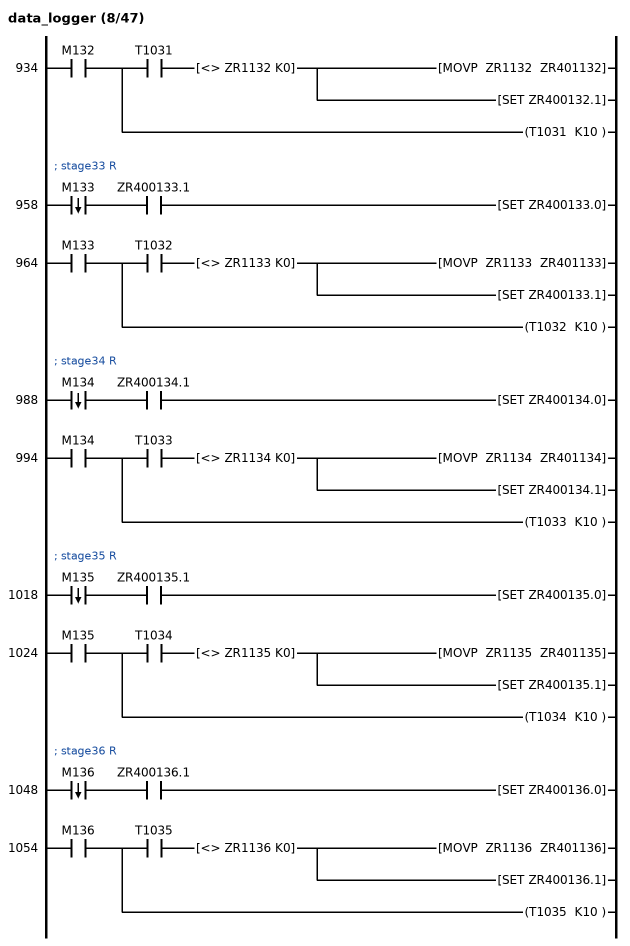
[picture p120: ladder of data_logger, rungs at steps 934 to 1054]
934   LD      M132
      MPS
      AND     T1031
      AND<>   ZR1132 K0
      MOVP    ZR1132 ZR401132
      SET     ZR400132.1
      MPP
      OUT     T1031 K10
; stage33 R
958   LDF     M133
      AND     ZR400133.1
      SET     ZR400133.0
964   LD      M133
      MPS
      AND     T1032
      AND<>   ZR1133 K0
      MOVP    ZR1133 ZR401133
      SET     ZR400133.1
      MPP
      OUT     T1032 K10
; stage34 R
988   LDF     M134
      AND     ZR400134.1
      SET     ZR400134.0
994   LD      M134
      MPS
      AND     T1033
      AND<>   ZR1134 K0
      MOVP    ZR1134 ZR401134
      SET     ZR400134.1
      MPP
      OUT     T1033 K10
; stage35 R
1018  LDF     M135
      AND     ZR400135.1
      SET     ZR400135.0
1024  LD      M135
      MPS
      AND     T1034
      AND<>   ZR1135 K0
      MOVP    ZR1135 ZR401135
      SET     ZR400135.1
      MPP
      OUT     T1034 K10
; stage36 R
1048  LDF     M136
      AND     ZR400136.1
      SET     ZR400136.0
1054  LD      M136
      MPS
      AND     T1035
      AND<>   ZR1136 K0
      MOVP    ZR1136 ZR401136
      SET     ZR400136.1
      MPP
      OUT     T1035 K10
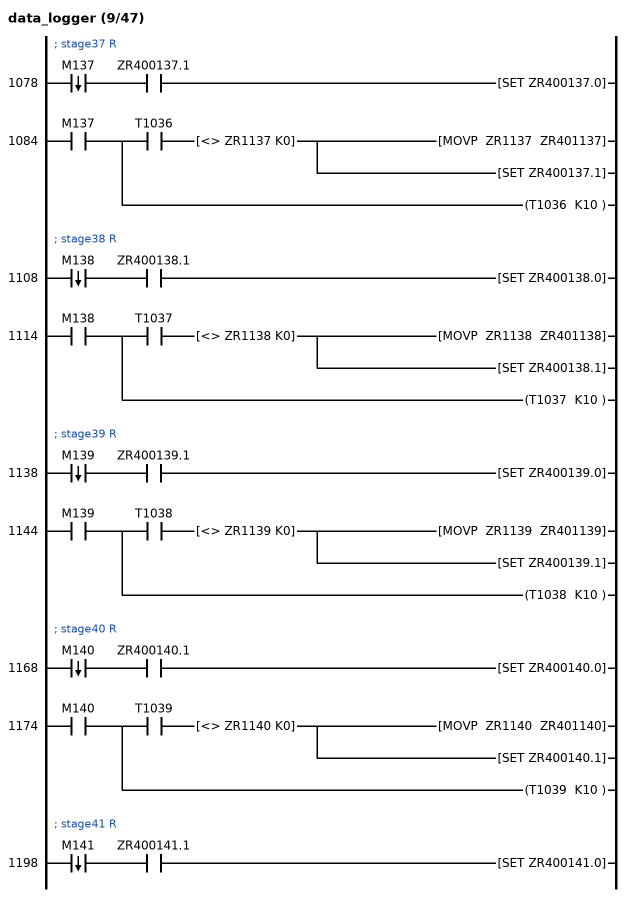
; stage37 R
1078  LDF     M137
      AND     ZR400137.1
      SET     ZR400137.0
1084  LD      M137
      MPS
      AND     T1036
      AND<>   ZR1137 K0
      MOVP    ZR1137 ZR401137
      SET     ZR400137.1
      MPP
      OUT     T1036 K10
; stage38 R
1108  LDF     M138
      AND     ZR400138.1
      SET     ZR400138.0
1114  LD      M138
      MPS
      AND     T1037
      AND<>   ZR1138 K0
      MOVP    ZR1138 ZR401138
      SET     ZR400138.1
      MPP
      OUT     T1037 K10
; stage39 R
1138  LDF     M139
      AND     ZR400139.1
      SET     ZR400139.0
1144  LD      M139
      MPS
      AND     T1038
      AND<>   ZR1139 K0
      MOVP    ZR1139 ZR401139
      SET     ZR400139.1
      MPP
      OUT     T1038 K10
; stage40 R
1168  LDF     M140
      AND     ZR400140.1
      SET     ZR400140.0
1174  LD      M140
      MPS
      AND     T1039
      AND<>   ZR1140 K0
      MOVP    ZR1140 ZR401140
      SET     ZR400140.1
      MPP
      OUT     T1039 K10
; stage41 R
1198  LDF     M141
      AND     ZR400141.1
      SET     ZR400141.0
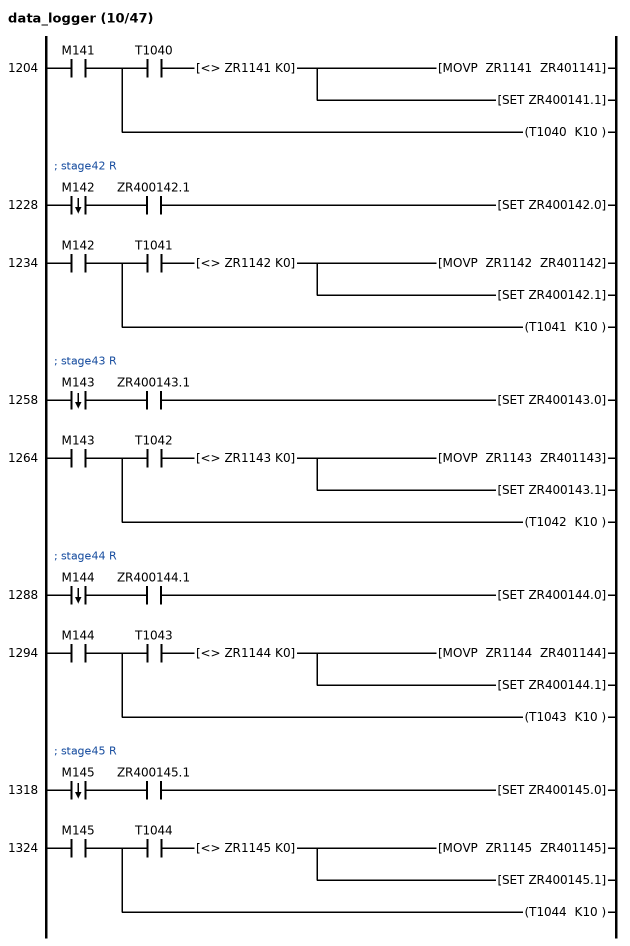
1204  LD      M141
      MPS
      AND     T1040
      AND<>   ZR1141 K0
      MOVP    ZR1141 ZR401141
      SET     ZR400141.1
      MPP
      OUT     T1040 K10
; stage42 R
1228  LDF     M142
      AND     ZR400142.1
      SET     ZR400142.0
1234  LD      M142
      MPS
      AND     T1041
      AND<>   ZR1142 K0
      MOVP    ZR1142 ZR401142
      SET     ZR400142.1
      MPP
      OUT     T1041 K10
; stage43 R
1258  LDF     M143
      AND     ZR400143.1
      SET     ZR400143.0
1264  LD      M143
      MPS
      AND     T1042
      AND<>   ZR1143 K0
      MOVP    ZR1143 ZR401143
      SET     ZR400143.1
      MPP
      OUT     T1042 K10
; stage44 R
1288  LDF     M144
      AND     ZR400144.1
      SET     ZR400144.0
1294  LD      M144
      MPS
      AND     T1043
      AND<>   ZR1144 K0
      MOVP    ZR1144 ZR401144
      SET     ZR400144.1
      MPP
      OUT     T1043 K10
; stage45 R
1318  LDF     M145
      AND     ZR400145.1
      SET     ZR400145.0
1324  LD      M145
      MPS
      AND     T1044
      AND<>   ZR1145 K0
      MOVP    ZR1145 ZR401145
      SET     ZR400145.1
      MPP
      OUT     T1044 K10
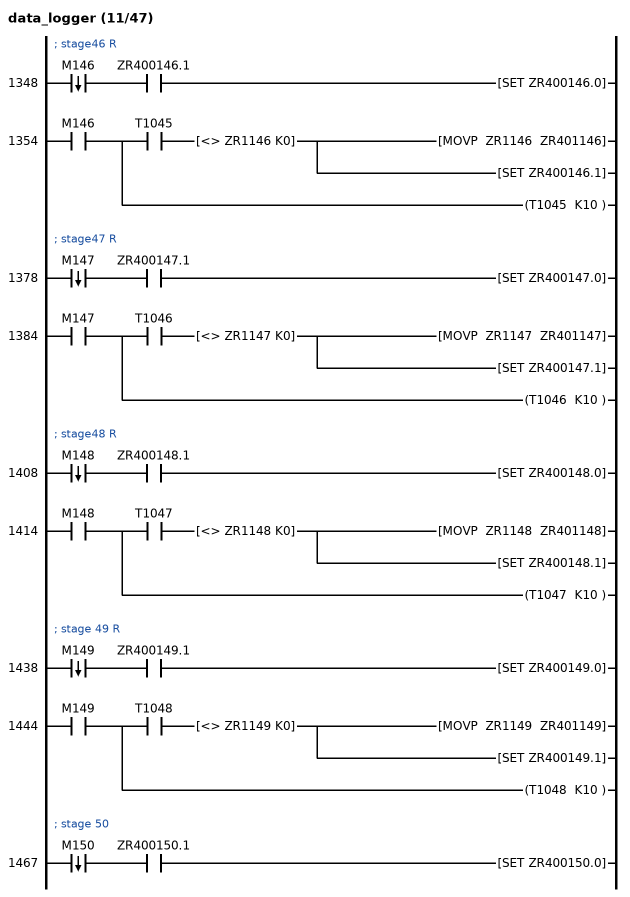
; stage46 R
1348  LDF     M146
      AND     ZR400146.1
      SET     ZR400146.0
1354  LD      M146
      MPS
      AND     T1045
      AND<>   ZR1146 K0
      MOVP    ZR1146 ZR401146
      SET     ZR400146.1
      MPP
      OUT     T1045 K10
; stage47 R
1378  LDF     M147
      AND     ZR400147.1
      SET     ZR400147.0
1384  LD      M147
      MPS
      AND     T1046
      AND<>   ZR1147 K0
      MOVP    ZR1147 ZR401147
      SET     ZR400147.1
      MPP
      OUT     T1046 K10
; stage48 R
1408  LDF     M148
      AND     ZR400148.1
      SET     ZR400148.0
1414  LD      M148
      MPS
      AND     T1047
      AND<>   ZR1148 K0
      MOVP    ZR1148 ZR401148
      SET     ZR400148.1
      MPP
      OUT     T1047 K10
; stage 49 R
1438  LDF     M149
      AND     ZR400149.1
      SET     ZR400149.0
1444  LD      M149
      MPS
      AND     T1048
      AND<>   ZR1149 K0
      MOVP    ZR1149 ZR401149
      SET     ZR400149.1
      MPP
      OUT     T1048 K10
; stage 50
1467  LDF     M150
      AND     ZR400150.1
      SET     ZR400150.0
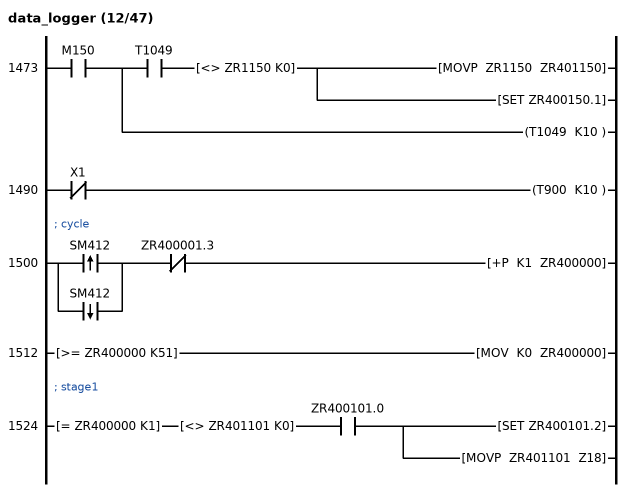
1473  LD      M150
      MPS
      AND     T1049
      AND<>   ZR1150 K0
      MOVP    ZR1150 ZR401150
      SET     ZR400150.1
      MPP
      OUT     T1049 K10
1490  LDI     X1
      OUT     T900 K10
; cycle
1500  LDP     SM412
      ORF     SM412
      ANI     ZR400001.3
      +P      K1 ZR400000
1512  LD>=    ZR400000 K51
      MOV     K0 ZR400000
; stage1
1524  LD=     ZR400000 K1
      AND<>   ZR401101 K0
      AND     ZR400101.0
      SET     ZR400101.2
      MOVP    ZR401101 Z18
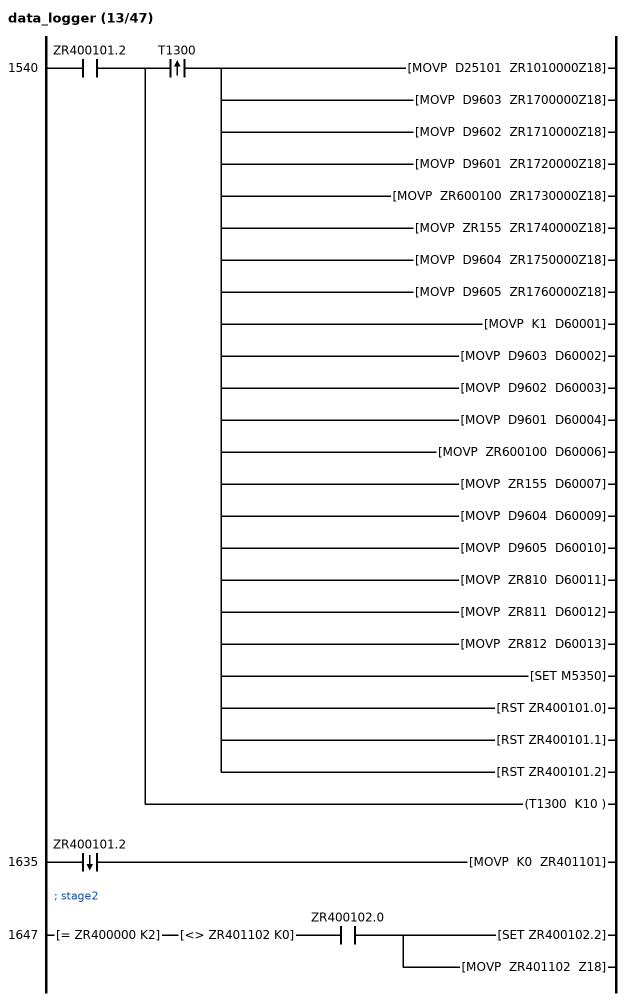
1540  LD      ZR400101.2
      MPS
      ANDP    T1300
      MOVP    D25101 ZR1010000Z18
      MOVP    D9603 ZR1700000Z18
      MOVP    D9602 ZR1710000Z18
      MOVP    D9601 ZR1720000Z18
      MOVP    ZR600100 ZR1730000Z18
      MOVP    ZR155 ZR1740000Z18
      MOVP    D9604 ZR1750000Z18
      MOVP    D9605 ZR1760000Z18
      MOVP    K1 D60001
      MOVP    D9603 D60002
      MOVP    D9602 D60003
      MOVP    D9601 D60004
      MOVP    ZR600100 D60006
      MOVP    ZR155 D60007
      MOVP    D9604 D60009
      MOVP    D9605 D60010
      MOVP    ZR810 D60011
      MOVP    ZR811 D60012
      MOVP    ZR812 D60013
      SET     M5350
      RST     ZR400101.0
      RST     ZR400101.1
      RST     ZR400101.2
      MPP
      OUT     T1300 K10
1635  LDF     ZR400101.2
      MOVP    K0 ZR401101
; stage2
1647  LD=     ZR400000 K2
      AND<>   ZR401102 K0
      AND     ZR400102.0
      SET     ZR400102.2
      MOVP    ZR401102 Z18
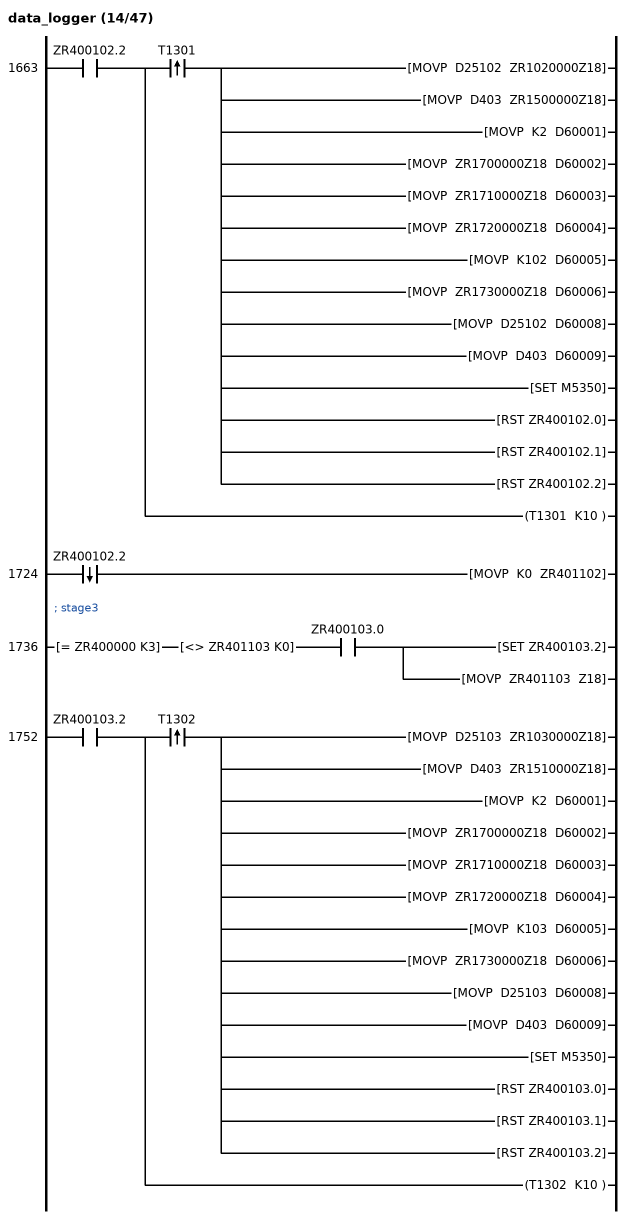
1663  LD      ZR400102.2
      MPS
      ANDP    T1301
      MOVP    D25102 ZR1020000Z18
      MOVP    D403 ZR1500000Z18
      MOVP    K2 D60001
      MOVP    ZR1700000Z18 D60002
      MOVP    ZR1710000Z18 D60003
      MOVP    ZR1720000Z18 D60004
      MOVP    K102 D60005
      MOVP    ZR1730000Z18 D60006
      MOVP    D25102 D60008
      MOVP    D403 D60009
      SET     M5350
      RST     ZR400102.0
      RST     ZR400102.1
      RST     ZR400102.2
      MPP
      OUT     T1301 K10
1724  LDF     ZR400102.2
      MOVP    K0 ZR401102
; stage3
1736  LD=     ZR400000 K3
      AND<>   ZR401103 K0
      AND     ZR400103.0
      SET     ZR400103.2
      MOVP    ZR401103 Z18
1752  LD      ZR400103.2
      MPS
      ANDP    T1302
      MOVP    D25103 ZR1030000Z18
      MOVP    D403 ZR1510000Z18
      MOVP    K2 D60001
      MOVP    ZR1700000Z18 D60002
      MOVP    ZR1710000Z18 D60003
      MOVP    ZR1720000Z18 D60004
      MOVP    K103 D60005
      MOVP    ZR1730000Z18 D60006
      MOVP    D25103 D60008
      MOVP    D403 D60009
      SET     M5350
      RST     ZR400103.0
      RST     ZR400103.1
      RST     ZR400103.2
      MPP
      OUT     T1302 K10
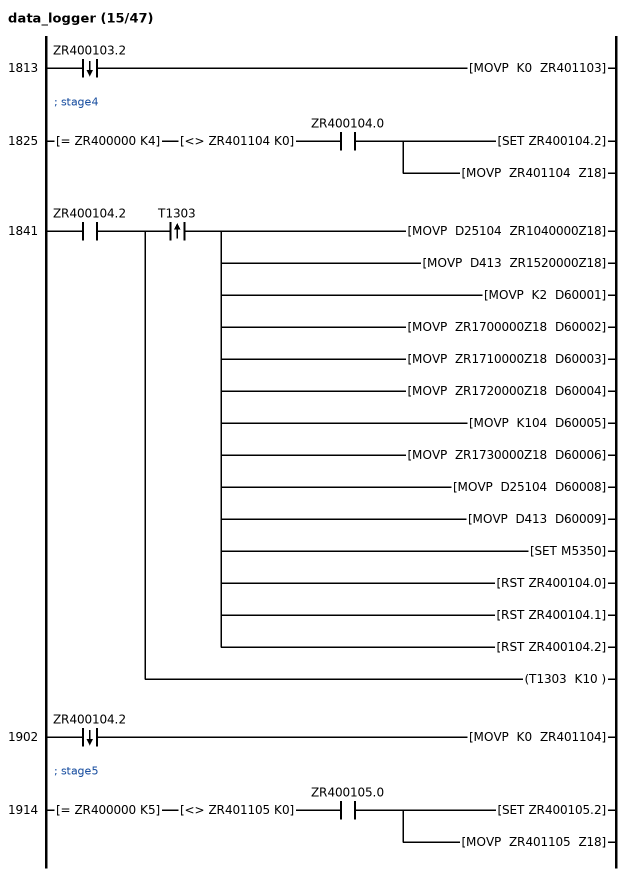
1813  LDF     ZR400103.2
      MOVP    K0 ZR401103
; stage4
1825  LD=     ZR400000 K4
      AND<>   ZR401104 K0
      AND     ZR400104.0
      SET     ZR400104.2
      MOVP    ZR401104 Z18
1841  LD      ZR400104.2
      MPS
      ANDP    T1303
      MOVP    D25104 ZR1040000Z18
      MOVP    D413 ZR1520000Z18
      MOVP    K2 D60001
      MOVP    ZR1700000Z18 D60002
      MOVP    ZR1710000Z18 D60003
      MOVP    ZR1720000Z18 D60004
      MOVP    K104 D60005
      MOVP    ZR1730000Z18 D60006
      MOVP    D25104 D60008
      MOVP    D413 D60009
      SET     M5350
      RST     ZR400104.0
      RST     ZR400104.1
      RST     ZR400104.2
      MPP
      OUT     T1303 K10
1902  LDF     ZR400104.2
      MOVP    K0 ZR401104
; stage5
1914  LD=     ZR400000 K5
      AND<>   ZR401105 K0
      AND     ZR400105.0
      SET     ZR400105.2
      MOVP    ZR401105 Z18
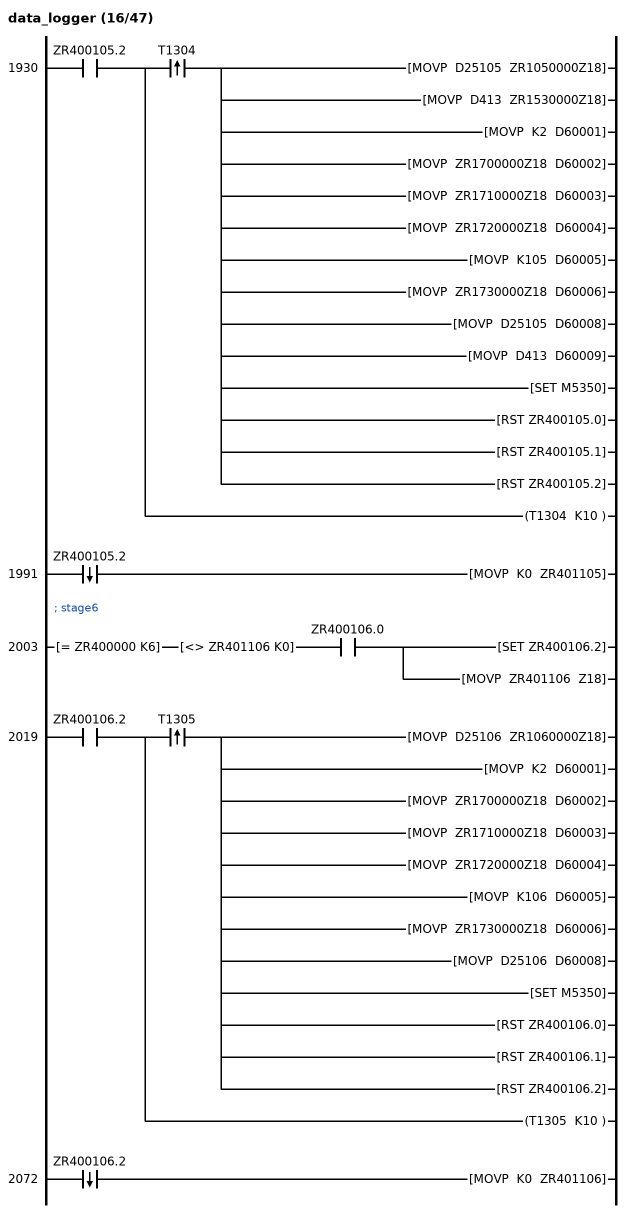
1930  LD      ZR400105.2
      MPS
      ANDP    T1304
      MOVP    D25105 ZR1050000Z18
      MOVP    D413 ZR1530000Z18
      MOVP    K2 D60001
      MOVP    ZR1700000Z18 D60002
      MOVP    ZR1710000Z18 D60003
      MOVP    ZR1720000Z18 D60004
      MOVP    K105 D60005
      MOVP    ZR1730000Z18 D60006
      MOVP    D25105 D60008
      MOVP    D413 D60009
      SET     M5350
      RST     ZR400105.0
      RST     ZR400105.1
      RST     ZR400105.2
      MPP
      OUT     T1304 K10
1991  LDF     ZR400105.2
      MOVP    K0 ZR401105
; stage6
2003  LD=     ZR400000 K6
      AND<>   ZR401106 K0
      AND     ZR400106.0
      SET     ZR400106.2
      MOVP    ZR401106 Z18
2019  LD      ZR400106.2
      MPS
      ANDP    T1305
      MOVP    D25106 ZR1060000Z18
      MOVP    K2 D60001
      MOVP    ZR1700000Z18 D60002
      MOVP    ZR1710000Z18 D60003
      MOVP    ZR1720000Z18 D60004
      MOVP    K106 D60005
      MOVP    ZR1730000Z18 D60006
      MOVP    D25106 D60008
      SET     M5350
      RST     ZR400106.0
      RST     ZR400106.1
      RST     ZR400106.2
      MPP
      OUT     T1305 K10
2072  LDF     ZR400106.2
      MOVP    K0 ZR401106
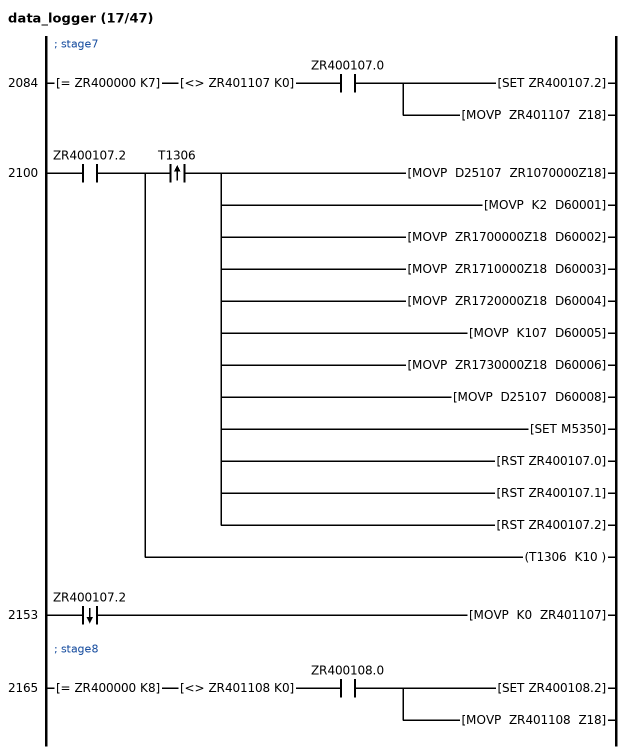
; stage7
2084  LD=     ZR400000 K7
      AND<>   ZR401107 K0
      AND     ZR400107.0
      SET     ZR400107.2
      MOVP    ZR401107 Z18
2100  LD      ZR400107.2
      MPS
      ANDP    T1306
      MOVP    D25107 ZR1070000Z18
      MOVP    K2 D60001
      MOVP    ZR1700000Z18 D60002
      MOVP    ZR1710000Z18 D60003
      MOVP    ZR1720000Z18 D60004
      MOVP    K107 D60005
      MOVP    ZR1730000Z18 D60006
      MOVP    D25107 D60008
      SET     M5350
      RST     ZR400107.0
      RST     ZR400107.1
      RST     ZR400107.2
      MPP
      OUT     T1306 K10
2153  LDF     ZR400107.2
      MOVP    K0 ZR401107
; stage8
2165  LD=     ZR400000 K8
      AND<>   ZR401108 K0
      AND     ZR400108.0
      SET     ZR400108.2
      MOVP    ZR401108 Z18
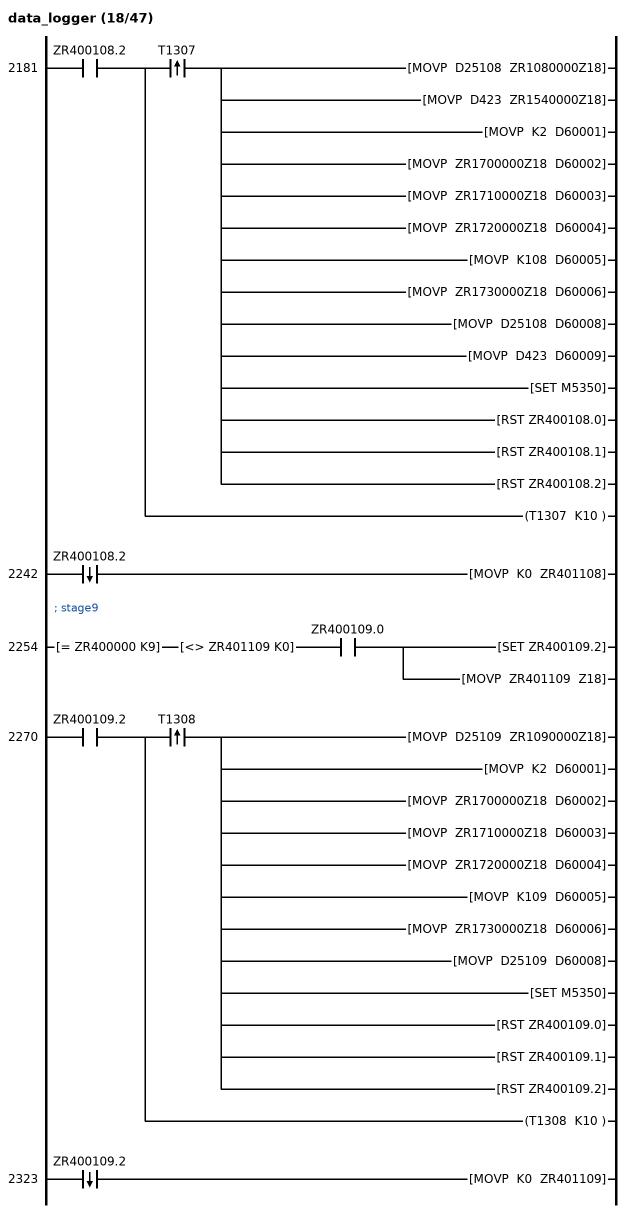
2181  LD      ZR400108.2
      MPS
      ANDP    T1307
      MOVP    D25108 ZR1080000Z18
      MOVP    D423 ZR1540000Z18
      MOVP    K2 D60001
      MOVP    ZR1700000Z18 D60002
      MOVP    ZR1710000Z18 D60003
      MOVP    ZR1720000Z18 D60004
      MOVP    K108 D60005
      MOVP    ZR1730000Z18 D60006
      MOVP    D25108 D60008
      MOVP    D423 D60009
      SET     M5350
      RST     ZR400108.0
      RST     ZR400108.1
      RST     ZR400108.2
      MPP
      OUT     T1307 K10
2242  LDF     ZR400108.2
      MOVP    K0 ZR401108
; stage9
2254  LD=     ZR400000 K9
      AND<>   ZR401109 K0
      AND     ZR400109.0
      SET     ZR400109.2
      MOVP    ZR401109 Z18
2270  LD      ZR400109.2
      MPS
      ANDP    T1308
      MOVP    D25109 ZR1090000Z18
      MOVP    K2 D60001
      MOVP    ZR1700000Z18 D60002
      MOVP    ZR1710000Z18 D60003
      MOVP    ZR1720000Z18 D60004
      MOVP    K109 D60005
      MOVP    ZR1730000Z18 D60006
      MOVP    D25109 D60008
      SET     M5350
      RST     ZR400109.0
      RST     ZR400109.1
      RST     ZR400109.2
      MPP
      OUT     T1308 K10
2323  LDF     ZR400109.2
      MOVP    K0 ZR401109
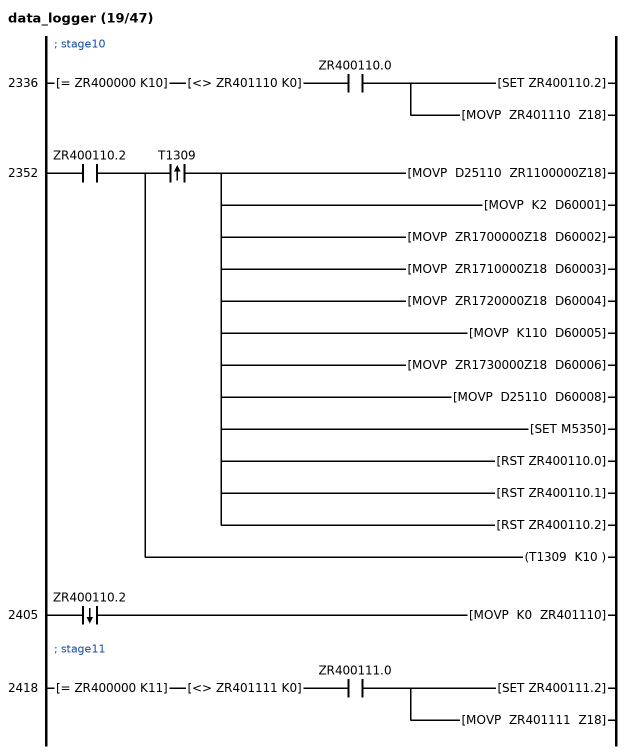
; stage10
2336  LD=     ZR400000 K10
      AND<>   ZR401110 K0
      AND     ZR400110.0
      SET     ZR400110.2
      MOVP    ZR401110 Z18
2352  LD      ZR400110.2
      MPS
      ANDP    T1309
      MOVP    D25110 ZR1100000Z18
      MOVP    K2 D60001
      MOVP    ZR1700000Z18 D60002
      MOVP    ZR1710000Z18 D60003
      MOVP    ZR1720000Z18 D60004
      MOVP    K110 D60005
      MOVP    ZR1730000Z18 D60006
      MOVP    D25110 D60008
      SET     M5350
      RST     ZR400110.0
      RST     ZR400110.1
      RST     ZR400110.2
      MPP
      OUT     T1309 K10
2405  LDF     ZR400110.2
      MOVP    K0 ZR401110
; stage11
2418  LD=     ZR400000 K11
      AND<>   ZR401111 K0
      AND     ZR400111.0
      SET     ZR400111.2
      MOVP    ZR401111 Z18
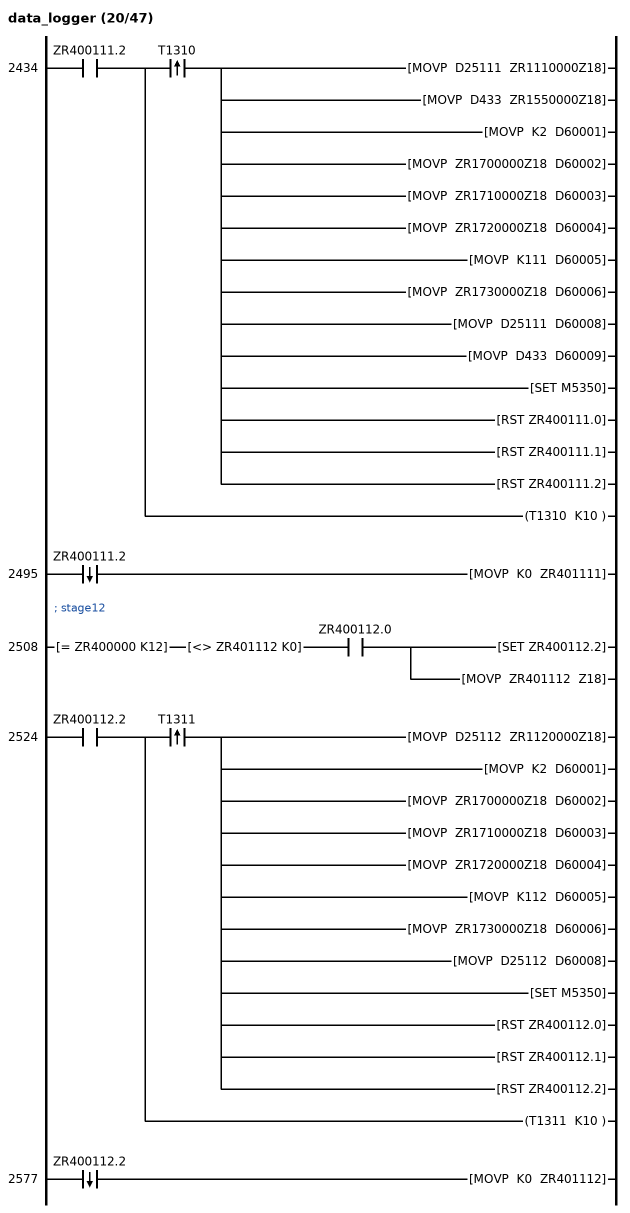
2434  LD      ZR400111.2
      MPS
      ANDP    T1310
      MOVP    D25111 ZR1110000Z18
      MOVP    D433 ZR1550000Z18
      MOVP    K2 D60001
      MOVP    ZR1700000Z18 D60002
      MOVP    ZR1710000Z18 D60003
      MOVP    ZR1720000Z18 D60004
      MOVP    K111 D60005
      MOVP    ZR1730000Z18 D60006
      MOVP    D25111 D60008
      MOVP    D433 D60009
      SET     M5350
      RST     ZR400111.0
      RST     ZR400111.1
      RST     ZR400111.2
      MPP
      OUT     T1310 K10
2495  LDF     ZR400111.2
      MOVP    K0 ZR401111
; stage12
2508  LD=     ZR400000 K12
      AND<>   ZR401112 K0
      AND     ZR400112.0
      SET     ZR400112.2
      MOVP    ZR401112 Z18
2524  LD      ZR400112.2
      MPS
      ANDP    T1311
      MOVP    D25112 ZR1120000Z18
      MOVP    K2 D60001
      MOVP    ZR1700000Z18 D60002
      MOVP    ZR1710000Z18 D60003
      MOVP    ZR1720000Z18 D60004
      MOVP    K112 D60005
      MOVP    ZR1730000Z18 D60006
      MOVP    D25112 D60008
      SET     M5350
      RST     ZR400112.0
      RST     ZR400112.1
      RST     ZR400112.2
      MPP
      OUT     T1311 K10
2577  LDF     ZR400112.2
      MOVP    K0 ZR401112
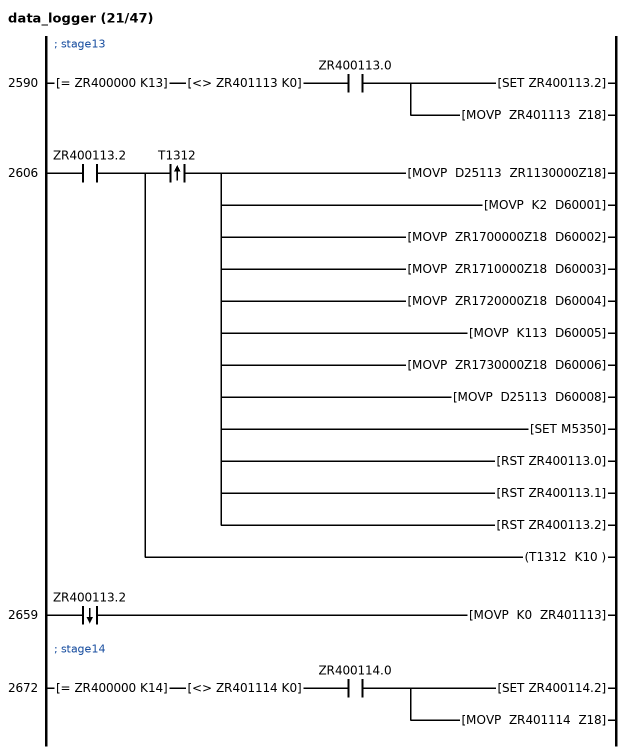
; stage13
2590  LD=     ZR400000 K13
      AND<>   ZR401113 K0
      AND     ZR400113.0
      SET     ZR400113.2
      MOVP    ZR401113 Z18
2606  LD      ZR400113.2
      MPS
      ANDP    T1312
      MOVP    D25113 ZR1130000Z18
      MOVP    K2 D60001
      MOVP    ZR1700000Z18 D60002
      MOVP    ZR1710000Z18 D60003
      MOVP    ZR1720000Z18 D60004
      MOVP    K113 D60005
      MOVP    ZR1730000Z18 D60006
      MOVP    D25113 D60008
      SET     M5350
      RST     ZR400113.0
      RST     ZR400113.1
      RST     ZR400113.2
      MPP
      OUT     T1312 K10
2659  LDF     ZR400113.2
      MOVP    K0 ZR401113
; stage14
2672  LD=     ZR400000 K14
      AND<>   ZR401114 K0
      AND     ZR400114.0
      SET     ZR400114.2
      MOVP    ZR401114 Z18
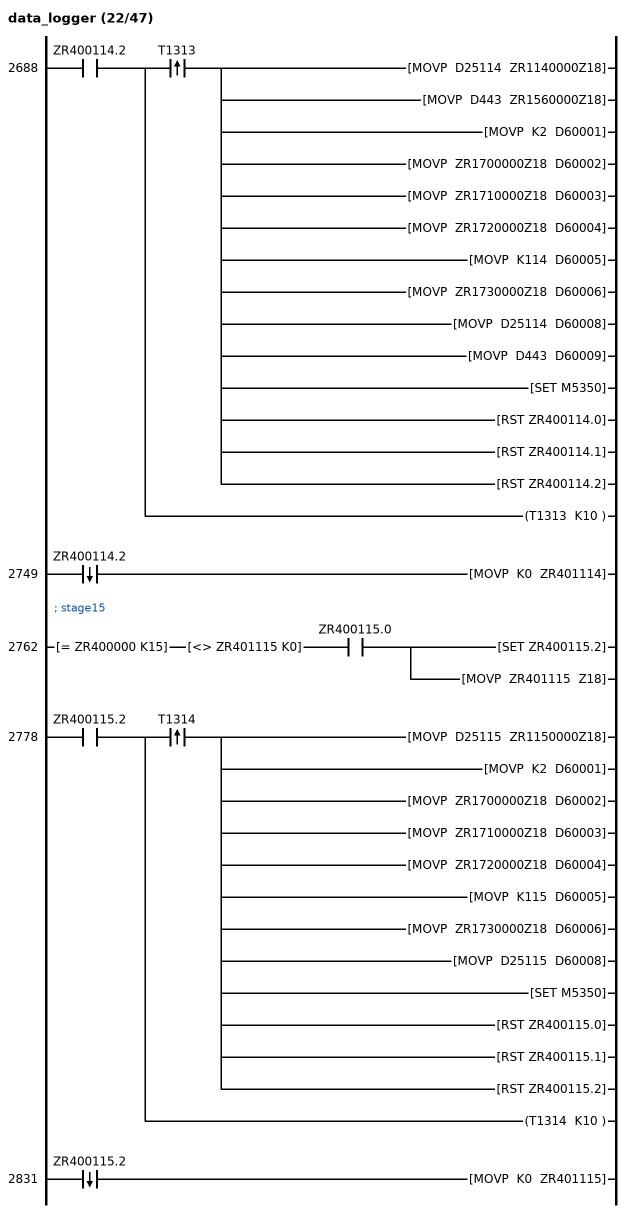
2688  LD      ZR400114.2
      MPS
      ANDP    T1313
      MOVP    D25114 ZR1140000Z18
      MOVP    D443 ZR1560000Z18
      MOVP    K2 D60001
      MOVP    ZR1700000Z18 D60002
      MOVP    ZR1710000Z18 D60003
      MOVP    ZR1720000Z18 D60004
      MOVP    K114 D60005
      MOVP    ZR1730000Z18 D60006
      MOVP    D25114 D60008
      MOVP    D443 D60009
      SET     M5350
      RST     ZR400114.0
      RST     ZR400114.1
      RST     ZR400114.2
      MPP
      OUT     T1313 K10
2749  LDF     ZR400114.2
      MOVP    K0 ZR401114
; stage15
2762  LD=     ZR400000 K15
      AND<>   ZR401115 K0
      AND     ZR400115.0
      SET     ZR400115.2
      MOVP    ZR401115 Z18
2778  LD      ZR400115.2
      MPS
      ANDP    T1314
      MOVP    D25115 ZR1150000Z18
      MOVP    K2 D60001
      MOVP    ZR1700000Z18 D60002
      MOVP    ZR1710000Z18 D60003
      MOVP    ZR1720000Z18 D60004
      MOVP    K115 D60005
      MOVP    ZR1730000Z18 D60006
      MOVP    D25115 D60008
      SET     M5350
      RST     ZR400115.0
      RST     ZR400115.1
      RST     ZR400115.2
      MPP
      OUT     T1314 K10
2831  LDF     ZR400115.2
      MOVP    K0 ZR401115
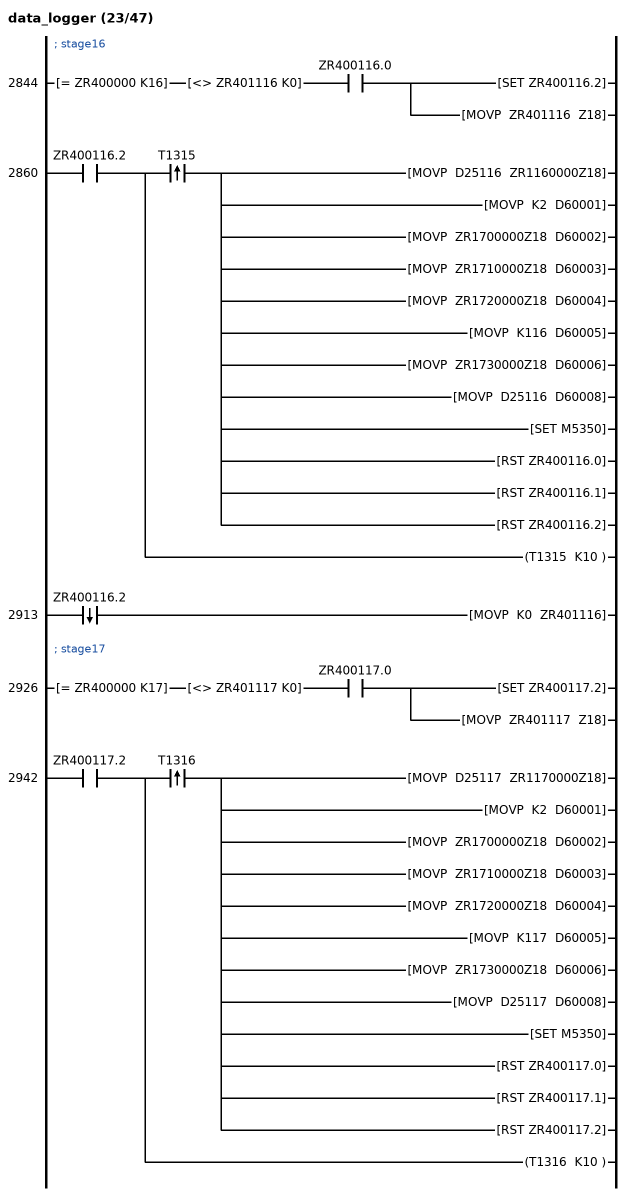
; stage16
2844  LD=     ZR400000 K16
      AND<>   ZR401116 K0
      AND     ZR400116.0
      SET     ZR400116.2
      MOVP    ZR401116 Z18
2860  LD      ZR400116.2
      MPS
      ANDP    T1315
      MOVP    D25116 ZR1160000Z18
      MOVP    K2 D60001
      MOVP    ZR1700000Z18 D60002
      MOVP    ZR1710000Z18 D60003
      MOVP    ZR1720000Z18 D60004
      MOVP    K116 D60005
      MOVP    ZR1730000Z18 D60006
      MOVP    D25116 D60008
      SET     M5350
      RST     ZR400116.0
      RST     ZR400116.1
      RST     ZR400116.2
      MPP
      OUT     T1315 K10
2913  LDF     ZR400116.2
      MOVP    K0 ZR401116
; stage17
2926  LD=     ZR400000 K17
      AND<>   ZR401117 K0
      AND     ZR400117.0
      SET     ZR400117.2
      MOVP    ZR401117 Z18
2942  LD      ZR400117.2
      MPS
      ANDP    T1316
      MOVP    D25117 ZR1170000Z18
      MOVP    K2 D60001
      MOVP    ZR1700000Z18 D60002
      MOVP    ZR1710000Z18 D60003
      MOVP    ZR1720000Z18 D60004
      MOVP    K117 D60005
      MOVP    ZR1730000Z18 D60006
      MOVP    D25117 D60008
      SET     M5350
      RST     ZR400117.0
      RST     ZR400117.1
      RST     ZR400117.2
      MPP
      OUT     T1316 K10
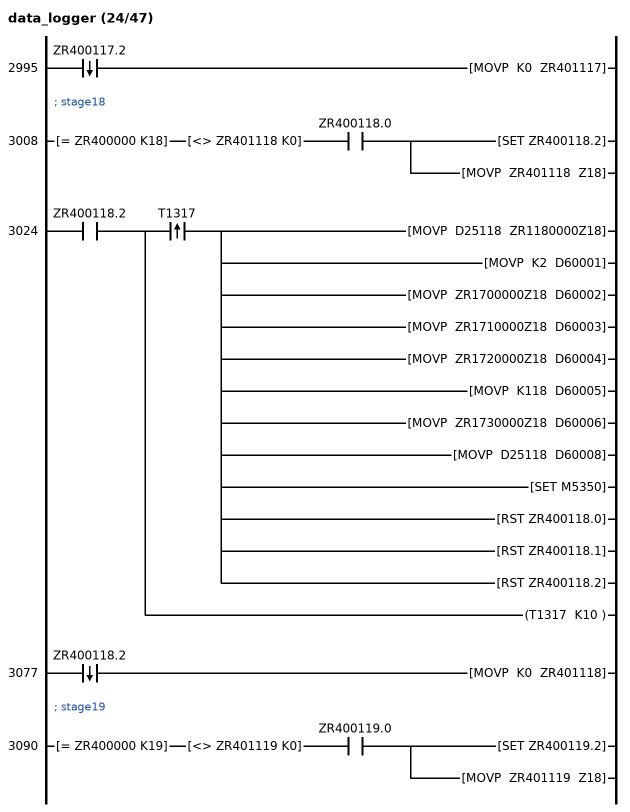
2995  LDF     ZR400117.2
      MOVP    K0 ZR401117
; stage18
3008  LD=     ZR400000 K18
      AND<>   ZR401118 K0
      AND     ZR400118.0
      SET     ZR400118.2
      MOVP    ZR401118 Z18
3024  LD      ZR400118.2
      MPS
      ANDP    T1317
      MOVP    D25118 ZR1180000Z18
      MOVP    K2 D60001
      MOVP    ZR1700000Z18 D60002
      MOVP    ZR1710000Z18 D60003
      MOVP    ZR1720000Z18 D60004
      MOVP    K118 D60005
      MOVP    ZR1730000Z18 D60006
      MOVP    D25118 D60008
      SET     M5350
      RST     ZR400118.0
      RST     ZR400118.1
      RST     ZR400118.2
      MPP
      OUT     T1317 K10
3077  LDF     ZR400118.2
      MOVP    K0 ZR401118
; stage19
3090  LD=     ZR400000 K19
      AND<>   ZR401119 K0
      AND     ZR400119.0
      SET     ZR400119.2
      MOVP    ZR401119 Z18
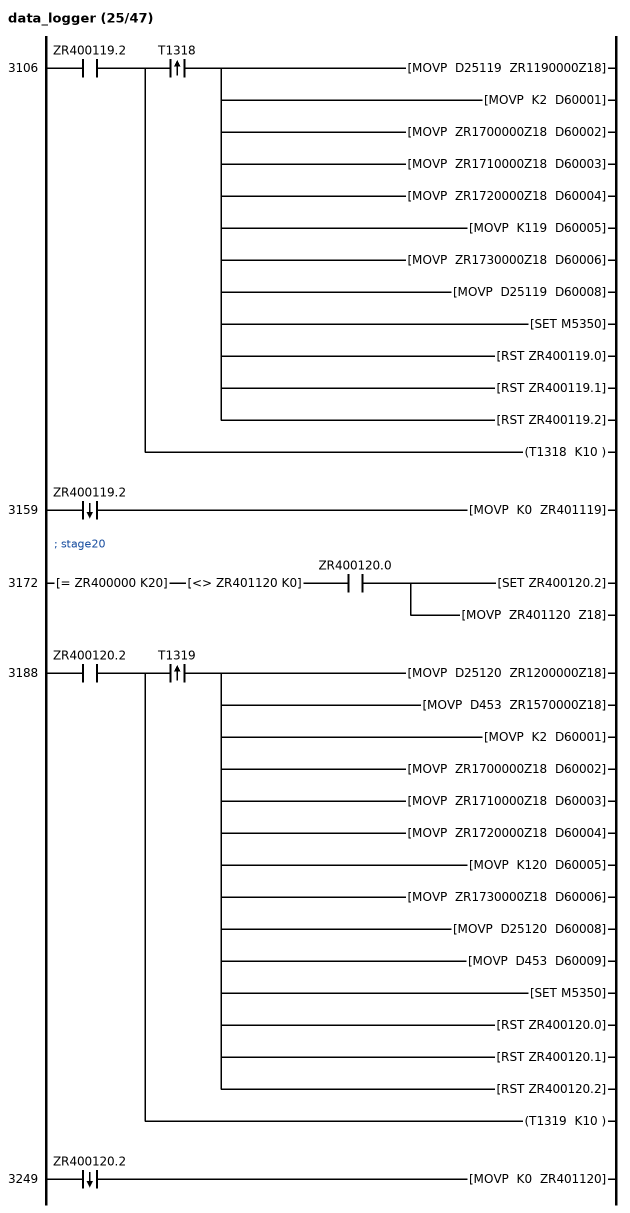
3106  LD      ZR400119.2
      MPS
      ANDP    T1318
      MOVP    D25119 ZR1190000Z18
      MOVP    K2 D60001
      MOVP    ZR1700000Z18 D60002
      MOVP    ZR1710000Z18 D60003
      MOVP    ZR1720000Z18 D60004
      MOVP    K119 D60005
      MOVP    ZR1730000Z18 D60006
      MOVP    D25119 D60008
      SET     M5350
      RST     ZR400119.0
      RST     ZR400119.1
      RST     ZR400119.2
      MPP
      OUT     T1318 K10
3159  LDF     ZR400119.2
      MOVP    K0 ZR401119
; stage20
3172  LD=     ZR400000 K20
      AND<>   ZR401120 K0
      AND     ZR400120.0
      SET     ZR400120.2
      MOVP    ZR401120 Z18
3188  LD      ZR400120.2
      MPS
      ANDP    T1319
      MOVP    D25120 ZR1200000Z18
      MOVP    D453 ZR1570000Z18
      MOVP    K2 D60001
      MOVP    ZR1700000Z18 D60002
      MOVP    ZR1710000Z18 D60003
      MOVP    ZR1720000Z18 D60004
      MOVP    K120 D60005
      MOVP    ZR1730000Z18 D60006
      MOVP    D25120 D60008
      MOVP    D453 D60009
      SET     M5350
      RST     ZR400120.0
      RST     ZR400120.1
      RST     ZR400120.2
      MPP
      OUT     T1319 K10
3249  LDF     ZR400120.2
      MOVP    K0 ZR401120
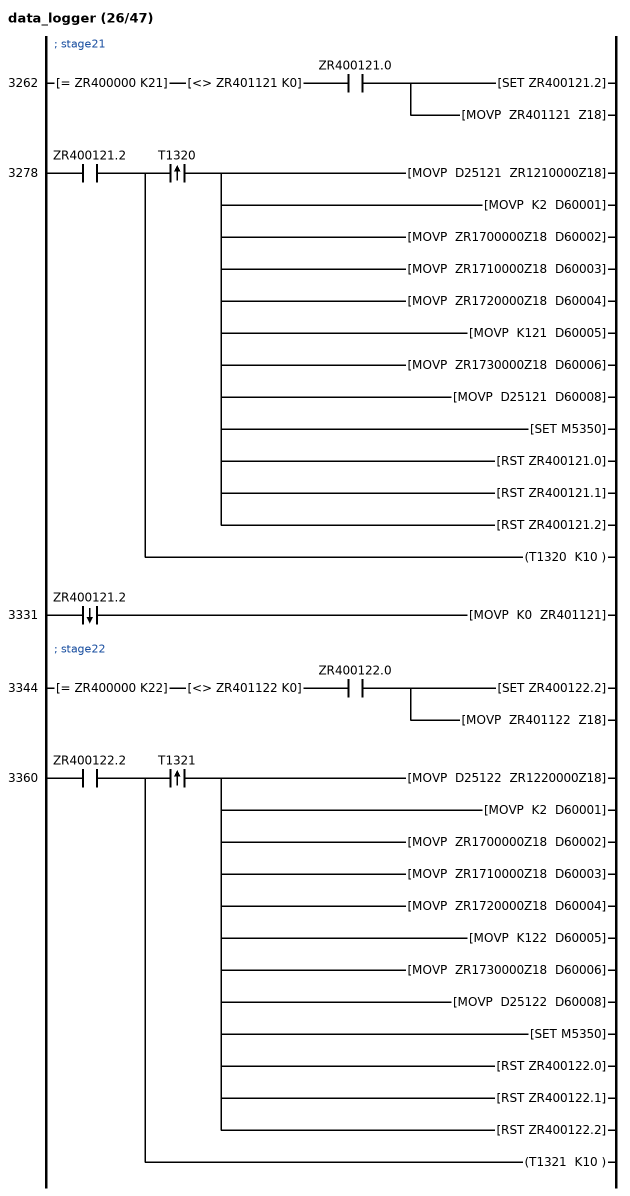
; stage21
3262  LD=     ZR400000 K21
      AND<>   ZR401121 K0
      AND     ZR400121.0
      SET     ZR400121.2
      MOVP    ZR401121 Z18
3278  LD      ZR400121.2
      MPS
      ANDP    T1320
      MOVP    D25121 ZR1210000Z18
      MOVP    K2 D60001
      MOVP    ZR1700000Z18 D60002
      MOVP    ZR1710000Z18 D60003
      MOVP    ZR1720000Z18 D60004
      MOVP    K121 D60005
      MOVP    ZR1730000Z18 D60006
      MOVP    D25121 D60008
      SET     M5350
      RST     ZR400121.0
      RST     ZR400121.1
      RST     ZR400121.2
      MPP
      OUT     T1320 K10
3331  LDF     ZR400121.2
      MOVP    K0 ZR401121
; stage22
3344  LD=     ZR400000 K22
      AND<>   ZR401122 K0
      AND     ZR400122.0
      SET     ZR400122.2
      MOVP    ZR401122 Z18
3360  LD      ZR400122.2
      MPS
      ANDP    T1321
      MOVP    D25122 ZR1220000Z18
      MOVP    K2 D60001
      MOVP    ZR1700000Z18 D60002
      MOVP    ZR1710000Z18 D60003
      MOVP    ZR1720000Z18 D60004
      MOVP    K122 D60005
      MOVP    ZR1730000Z18 D60006
      MOVP    D25122 D60008
      SET     M5350
      RST     ZR400122.0
      RST     ZR400122.1
      RST     ZR400122.2
      MPP
      OUT     T1321 K10
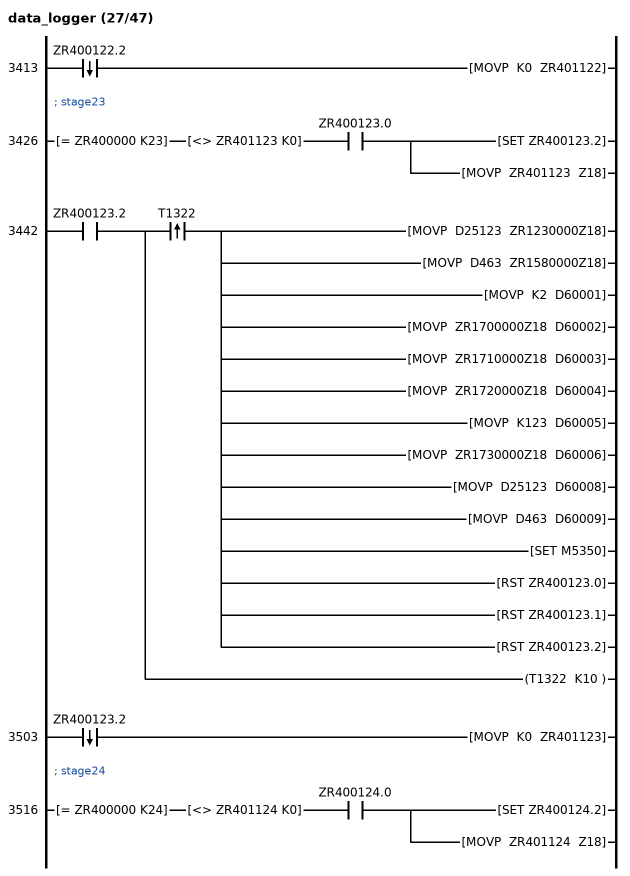
3413  LDF     ZR400122.2
      MOVP    K0 ZR401122
; stage23
3426  LD=     ZR400000 K23
      AND<>   ZR401123 K0
      AND     ZR400123.0
      SET     ZR400123.2
      MOVP    ZR401123 Z18
3442  LD      ZR400123.2
      MPS
      ANDP    T1322
      MOVP    D25123 ZR1230000Z18
      MOVP    D463 ZR1580000Z18
      MOVP    K2 D60001
      MOVP    ZR1700000Z18 D60002
      MOVP    ZR1710000Z18 D60003
      MOVP    ZR1720000Z18 D60004
      MOVP    K123 D60005
      MOVP    ZR1730000Z18 D60006
      MOVP    D25123 D60008
      MOVP    D463 D60009
      SET     M5350
      RST     ZR400123.0
      RST     ZR400123.1
      RST     ZR400123.2
      MPP
      OUT     T1322 K10
3503  LDF     ZR400123.2
      MOVP    K0 ZR401123
; stage24
3516  LD=     ZR400000 K24
      AND<>   ZR401124 K0
      AND     ZR400124.0
      SET     ZR400124.2
      MOVP    ZR401124 Z18
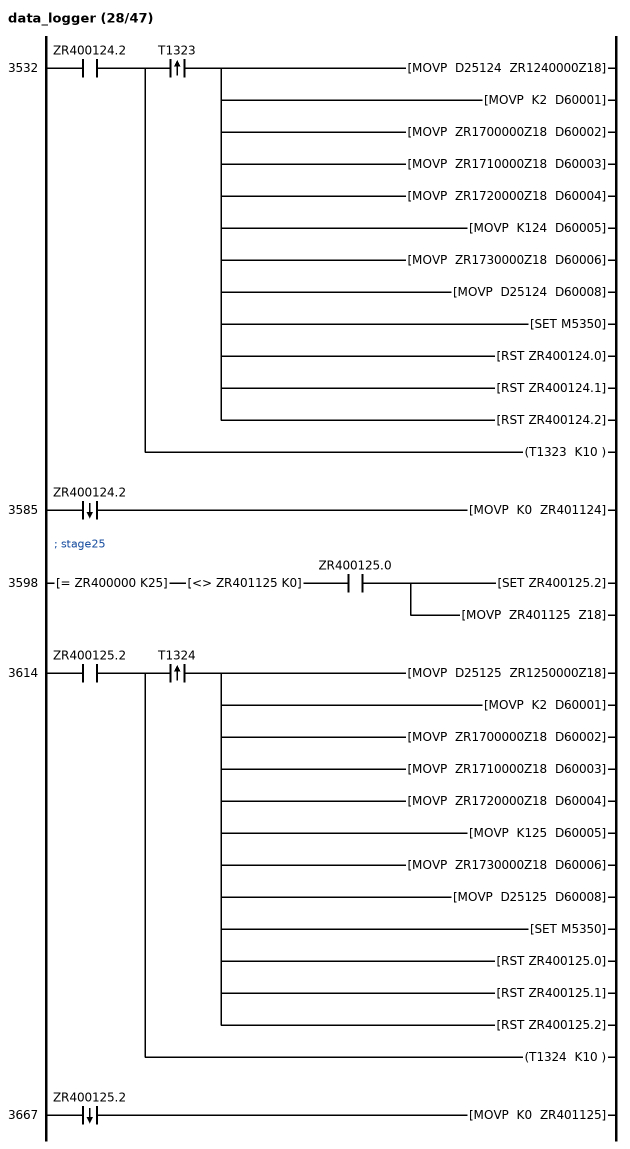
3532  LD      ZR400124.2
      MPS
      ANDP    T1323
      MOVP    D25124 ZR1240000Z18
      MOVP    K2 D60001
      MOVP    ZR1700000Z18 D60002
      MOVP    ZR1710000Z18 D60003
      MOVP    ZR1720000Z18 D60004
      MOVP    K124 D60005
      MOVP    ZR1730000Z18 D60006
      MOVP    D25124 D60008
      SET     M5350
      RST     ZR400124.0
      RST     ZR400124.1
      RST     ZR400124.2
      MPP
      OUT     T1323 K10
3585  LDF     ZR400124.2
      MOVP    K0 ZR401124
; stage25
3598  LD=     ZR400000 K25
      AND<>   ZR401125 K0
      AND     ZR400125.0
      SET     ZR400125.2
      MOVP    ZR401125 Z18
3614  LD      ZR400125.2
      MPS
      ANDP    T1324
      MOVP    D25125 ZR1250000Z18
      MOVP    K2 D60001
      MOVP    ZR1700000Z18 D60002
      MOVP    ZR1710000Z18 D60003
      MOVP    ZR1720000Z18 D60004
      MOVP    K125 D60005
      MOVP    ZR1730000Z18 D60006
      MOVP    D25125 D60008
      SET     M5350
      RST     ZR400125.0
      RST     ZR400125.1
      RST     ZR400125.2
      MPP
      OUT     T1324 K10
3667  LDF     ZR400125.2
      MOVP    K0 ZR401125
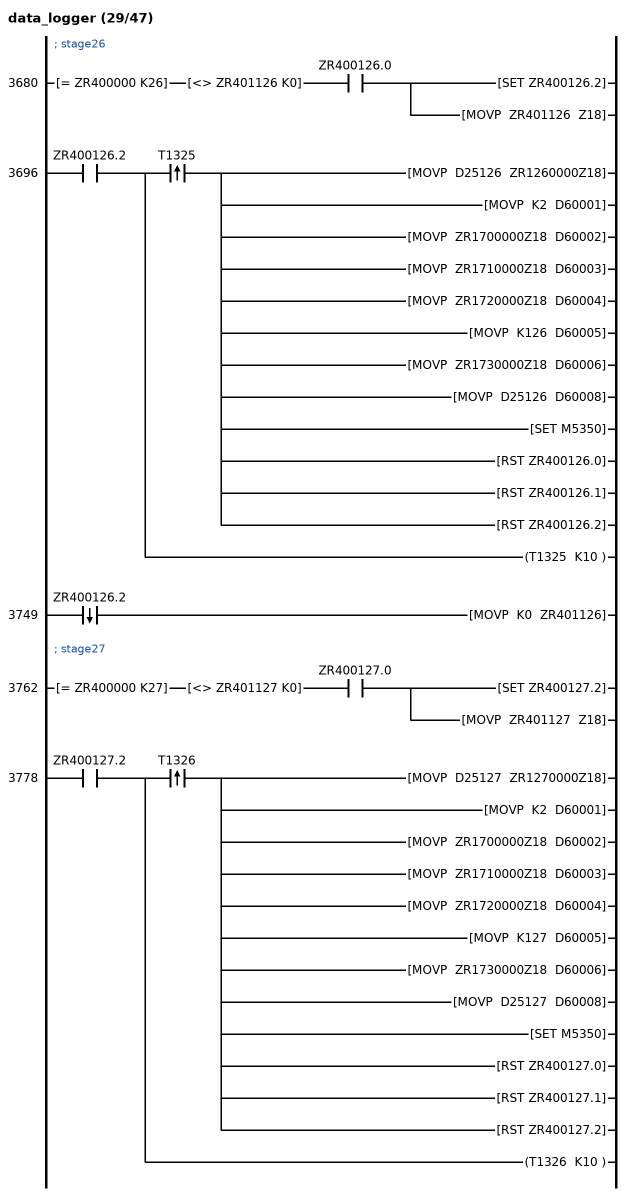
; stage26
3680  LD=     ZR400000 K26
      AND<>   ZR401126 K0
      AND     ZR400126.0
      SET     ZR400126.2
      MOVP    ZR401126 Z18
3696  LD      ZR400126.2
      MPS
      ANDP    T1325
      MOVP    D25126 ZR1260000Z18
      MOVP    K2 D60001
      MOVP    ZR1700000Z18 D60002
      MOVP    ZR1710000Z18 D60003
      MOVP    ZR1720000Z18 D60004
      MOVP    K126 D60005
      MOVP    ZR1730000Z18 D60006
      MOVP    D25126 D60008
      SET     M5350
      RST     ZR400126.0
      RST     ZR400126.1
      RST     ZR400126.2
      MPP
      OUT     T1325 K10
3749  LDF     ZR400126.2
      MOVP    K0 ZR401126
; stage27
3762  LD=     ZR400000 K27
      AND<>   ZR401127 K0
      AND     ZR400127.0
      SET     ZR400127.2
      MOVP    ZR401127 Z18
3778  LD      ZR400127.2
      MPS
      ANDP    T1326
      MOVP    D25127 ZR1270000Z18
      MOVP    K2 D60001
      MOVP    ZR1700000Z18 D60002
      MOVP    ZR1710000Z18 D60003
      MOVP    ZR1720000Z18 D60004
      MOVP    K127 D60005
      MOVP    ZR1730000Z18 D60006
      MOVP    D25127 D60008
      SET     M5350
      RST     ZR400127.0
      RST     ZR400127.1
      RST     ZR400127.2
      MPP
      OUT     T1326 K10
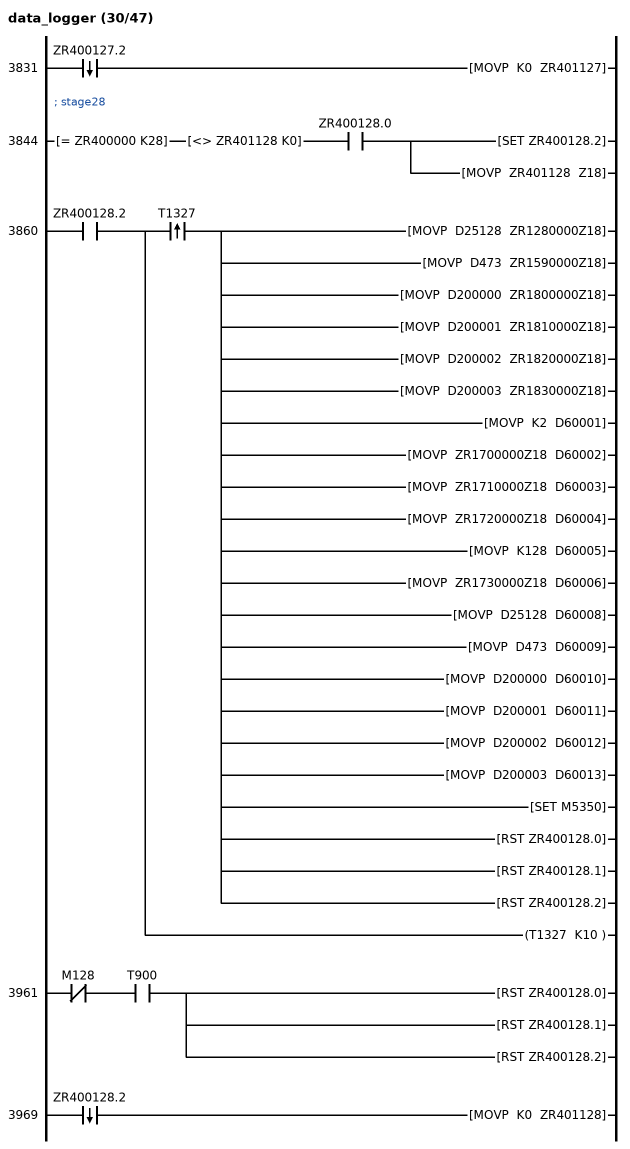
3831  LDF     ZR400127.2
      MOVP    K0 ZR401127
; stage28
3844  LD=     ZR400000 K28
      AND<>   ZR401128 K0
      AND     ZR400128.0
      SET     ZR400128.2
      MOVP    ZR401128 Z18
3860  LD      ZR400128.2
      MPS
      ANDP    T1327
      MOVP    D25128 ZR1280000Z18
      MOVP    D473 ZR1590000Z18
      MOVP    D200000 ZR1800000Z18
      MOVP    D200001 ZR1810000Z18
      MOVP    D200002 ZR1820000Z18
      MOVP    D200003 ZR1830000Z18
      MOVP    K2 D60001
      MOVP    ZR1700000Z18 D60002
      MOVP    ZR1710000Z18 D60003
      MOVP    ZR1720000Z18 D60004
      MOVP    K128 D60005
      MOVP    ZR1730000Z18 D60006
      MOVP    D25128 D60008
      MOVP    D473 D60009
      MOVP    D200000 D60010
      MOVP    D200001 D60011
      MOVP    D200002 D60012
      MOVP    D200003 D60013
      SET     M5350
      RST     ZR400128.0
      RST     ZR400128.1
      RST     ZR400128.2
      MPP
      OUT     T1327 K10
3961  LDI     M128
      AND     T900
      RST     ZR400128.0
      RST     ZR400128.1
      RST     ZR400128.2
3969  LDF     ZR400128.2
      MOVP    K0 ZR401128
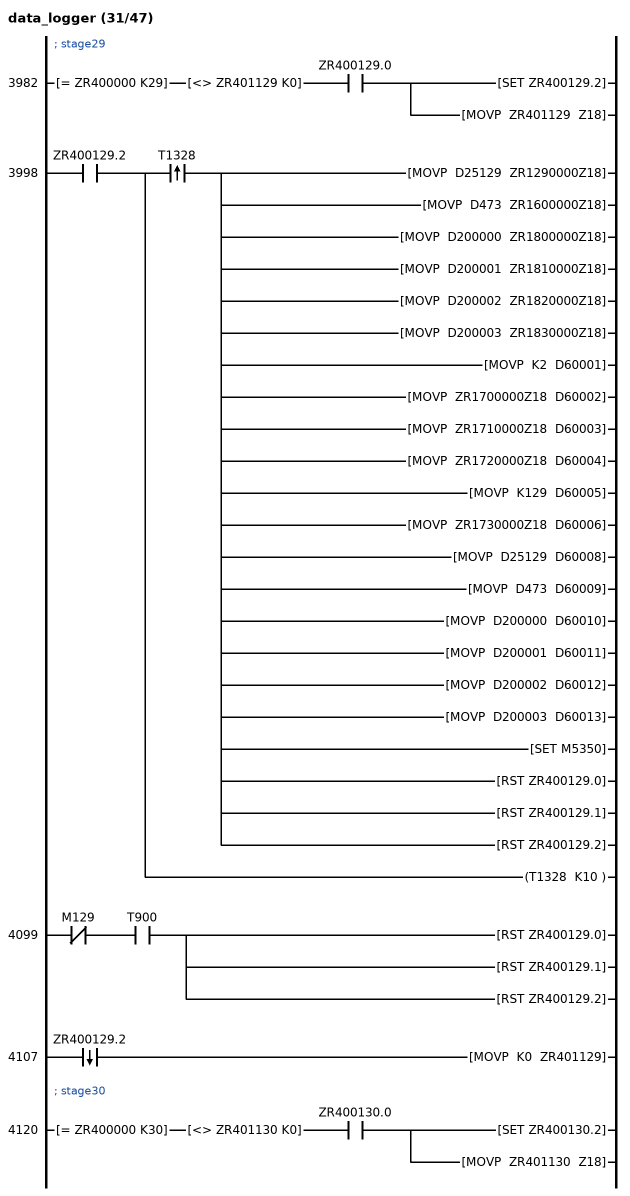
; stage29
3982  LD=     ZR400000 K29
      AND<>   ZR401129 K0
      AND     ZR400129.0
      SET     ZR400129.2
      MOVP    ZR401129 Z18
3998  LD      ZR400129.2
      MPS
      ANDP    T1328
      MOVP    D25129 ZR1290000Z18
      MOVP    D473 ZR1600000Z18
      MOVP    D200000 ZR1800000Z18
      MOVP    D200001 ZR1810000Z18
      MOVP    D200002 ZR1820000Z18
      MOVP    D200003 ZR1830000Z18
      MOVP    K2 D60001
      MOVP    ZR1700000Z18 D60002
      MOVP    ZR1710000Z18 D60003
      MOVP    ZR1720000Z18 D60004
      MOVP    K129 D60005
      MOVP    ZR1730000Z18 D60006
      MOVP    D25129 D60008
      MOVP    D473 D60009
      MOVP    D200000 D60010
      MOVP    D200001 D60011
      MOVP    D200002 D60012
      MOVP    D200003 D60013
      SET     M5350
      RST     ZR400129.0
      RST     ZR400129.1
      RST     ZR400129.2
      MPP
      OUT     T1328 K10
4099  LDI     M129
      AND     T900
      RST     ZR400129.0
      RST     ZR400129.1
      RST     ZR400129.2
4107  LDF     ZR400129.2
      MOVP    K0 ZR401129
; stage30
4120  LD=     ZR400000 K30
      AND<>   ZR401130 K0
      AND     ZR400130.0
      SET     ZR400130.2
      MOVP    ZR401130 Z18
